TYPE ST_LaudaReadCommands_Status :
STRUCT
	StandBy			: STRING := 'IN_MODE_02';
	DeviceType		: STRING := 'TYPE';
	DeviceStatus	: STRING := 'STATUS';
	FaultDiagnosis	: STRING := 'STAT';
	
END_STRUCT
END_TYPE

(* stored: Version 1.1.0.1, ProductVersion 3.1.4024.12
   DUT ST_LaudaReadCommands_Status: Id {cc79e912-c922-4b78-80c1-e387294f653c} *)
